FUNCTION TryConvert_BOOL_TO_DINT : BOOL
VAR_INPUT
	in : BOOL;
	out : REFERENCE TO DINT;
END_VAR

out := BOOL_TO_DINT(in);
TryConvert_BOOL_TO_DINT := TRUE;

END_FUNCTION

(* stored: Version 1.1.0.1, ProductVersion 3.1.4024.12
   POU TryConvert_BOOL_TO_DINT: Id {a764e9d8-9af9-4541-b414-cc28c823458a}, SpecialFunc None *)
